{attribute 'qualified_only'}
VAR_GLOBAL
	fSpeedToleranceRpm: LREAL := 0.05;
	
END_VAR

VAR_GLOBAL CONSTANT
	nSectors: LREAL :=36;
    nPulseFreqHz:LREAL:=14;
	fNominalSpeedRpm: LREAL := Target_GlobalVariableList.nPulseFreqHz/Target_GlobalVariableList.nSectors*60;
    fMaximumSPeedRpm: LREAL := Target_GlobalVariableList.fNominalSpeedRpm*1.1;
	nMaxMotorTemperature: INT:= 80;
	fWheelDiameter:LREAL:=2500;
	//ErrorCodes
	nErrorIdNoLatch:INT:=1000;
END_VAR

(* stored: Version 1.1.0.1, ProductVersion 3.1.4022.6
   GVL Target_GlobalVariableList: Id {c7b465dd-090c-4ea5-b2d2-91bf4a0ef82f} *)
